FUNCTION Call_HMI

//hmiOperatingmodeInterface.PLCToHMI.CurrentOperatingMode := instOperatingMode.StateOperatingMode;
hmiHeaderInstance(NameApplication := 'Hochregallager',
				  OperatingModeHMIInterface := hmiOperatingmodeInterface,
				  HeaderHMIInterface := hmiHeaderInterface);
				  
hmiAdsCommunicationInterfaceInstance(Timeout := T#1S,
									 TimeoutHMI := T#500ms,
									 LocalAdsPort := 851,
									 HeartbeatHMI := hmiAdsCommunicationInterface.HeartbeatHMI);
									 

hmiAdsCommunicationInterface.DeviceIpAddress := hmiAdsCommunicationInterfaceInstance.LocalIpAddress;
hmiAdsCommunicationInterface.LocalAMSNetId := hmiAdsCommunicationInterfaceInstance.LocalAMSNetId;
hmiAdsCommunicationInterface.HeartbeatPLC := hmiAdsCommunicationInterfaceInstance.PLCHeartbeatHMICommunication;
hmiAdsCommunicationInterface.RuntimeStatus := hmiAdsCommunicationInterfaceInstance.AdsState;

// FC_InitializingSettingLines(HMIInterface := HMI.hmiMachineSectionInterface);

END_FUNCTION

(* stored: Version 1.1.0.1
   POU Call_HMI: Id {619c281c-ef5d-4639-891a-10e7108f6cf6}, SpecialFunc None *)
